Universal Robots PolyScope program: URCap.urp

Program URCap (installation=docker directory=/ursim/programs createdIn=3.15.8.106339 lastSavedIn=3.15.8.106339 robotSerialNumber=2018309999)
Calibrated DH parameters: a=[0, -0.612, -0.5723, 0, 0, 0]; d=[0.1273, 0, 0, 0.163941, 0.1157, 0.0922]; alpha=[1.570796, 0, 0, 1.570796, -1.570796, 0]; deltaTheta=[0, 0, 0, 0, 0, 0]
Robot Program (runOnlyOnce=false)
  URCap External Control (External Control, FZI Research Center for Information Technology)
